{attribute 'qualified_only'}
{attribute 'strict'}
TYPE E_Message_PV :
(
	eNoMessage := 0,
	eTooMuchPV := 1,
	ePvError := 2,
	eNoConnectionToBackend := 3
);
END_TYPE

(* stored: Version 1.1.0.1, ProductVersion 3.1.4024.6
   DUT E_Message_PV: Id {1d99da9e-c517-47e3-9ee7-cb34eba93936} *)
